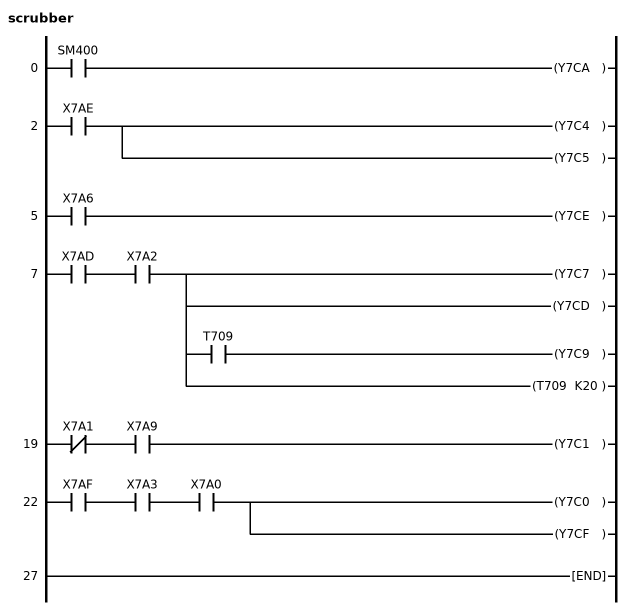
[picture p192: ladder of scrubber, rungs at steps 0 to 27]
0     LD      SM400
      OUT     Y7CA
2     LD      X7AE
      OUT     Y7C4
      OUT     Y7C5
5     LD      X7A6
      OUT     Y7CE
7     LD      X7AD
      AND     X7A2
      OUT     Y7C7
      OUT     Y7CD
      MPS
      AND     T709
      OUT     Y7C9
      MPP
      OUT     T709 K20
19    LDI     X7A1
      AND     X7A9
      OUT     Y7C1
22    LD      X7AF
      AND     X7A3
      AND     X7A0
      OUT     Y7C0
      OUT     Y7CF
27    END
END_PROGRAM

PROGRAM send_to_c
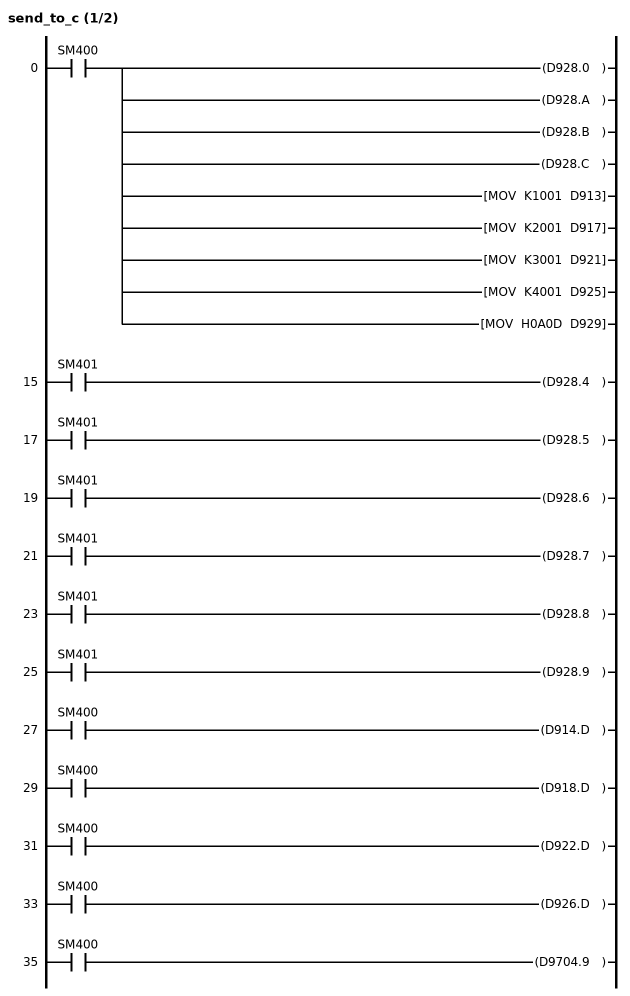
0     LD      SM400
      OUT     D928.0
      OUT     D928.A
      OUT     D928.B
      OUT     D928.C
      MOV     K1001 D913
      MOV     K2001 D917
      MOV     K3001 D921
      MOV     K4001 D925
      MOV     H0A0D D929
15    LD      SM401
      OUT     D928.4
17    LD      SM401
      OUT     D928.5
19    LD      SM401
      OUT     D928.6
21    LD      SM401
      OUT     D928.7
23    LD      SM401
      OUT     D928.8
25    LD      SM401
      OUT     D928.9
27    LD      SM400
      OUT     D914.D
29    LD      SM400
      OUT     D918.D
31    LD      SM400
      OUT     D922.D
33    LD      SM400
      OUT     D926.D
35    LD      SM400
      OUT     D9704.9
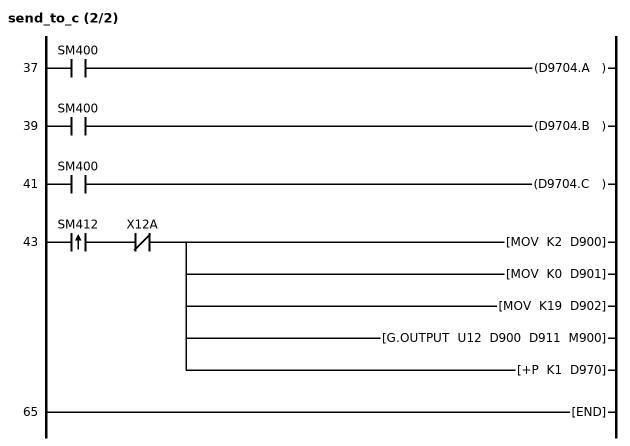
37    LD      SM400
      OUT     D9704.A
39    LD      SM400
      OUT     D9704.B
41    LD      SM400
      OUT     D9704.C
43    LDP     SM412
      ANI     X12A
      MOV     K2 D900
      MOV     K0 D901
      MOV     K19 D902
      G.OUTPUT U12 D900 D911 M900
      +P      K1 D970
65    END
END_PROGRAM

PROGRAM shower
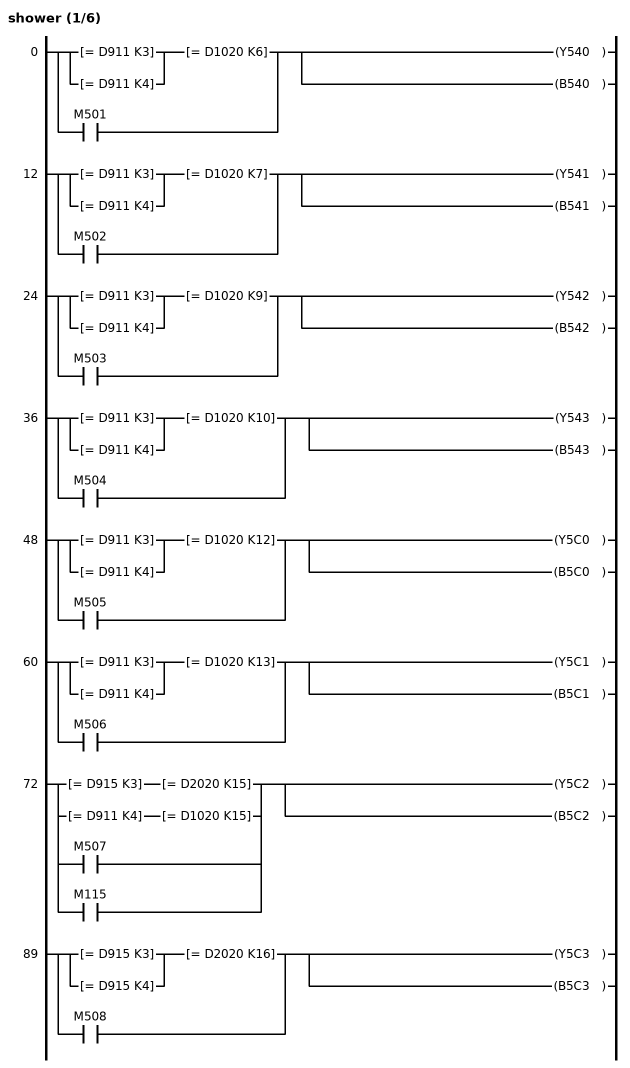
0     LD=     D911 K3
      OR=     D911 K4
      AND=    D1020 K6
      OR      M501
      OUT     Y540
      OUT     B540
12    LD=     D911 K3
      OR=     D911 K4
      AND=    D1020 K7
      OR      M502
      OUT     Y541
      OUT     B541
24    LD=     D911 K3
      OR=     D911 K4
      AND=    D1020 K9
      OR      M503
      OUT     Y542
      OUT     B542
36    LD=     D911 K3
      OR=     D911 K4
      AND=    D1020 K10
      OR      M504
      OUT     Y543
      OUT     B543
48    LD=     D911 K3
      OR=     D911 K4
      AND=    D1020 K12
      OR      M505
      OUT     Y5C0
      OUT     B5C0
60    LD=     D911 K3
      OR=     D911 K4
      AND=    D1020 K13
      OR      M506
      OUT     Y5C1
      OUT     B5C1
72    LD=     D915 K3
      AND=    D2020 K15
      LD=     D911 K4
      AND=    D1020 K15
      ORB
      OR      M507
      OR      M115
      OUT     Y5C2
      OUT     B5C2
89    LD=     D915 K3
      OR=     D915 K4
      AND=    D2020 K16
      OR      M508
      OUT     Y5C3
      OUT     B5C3
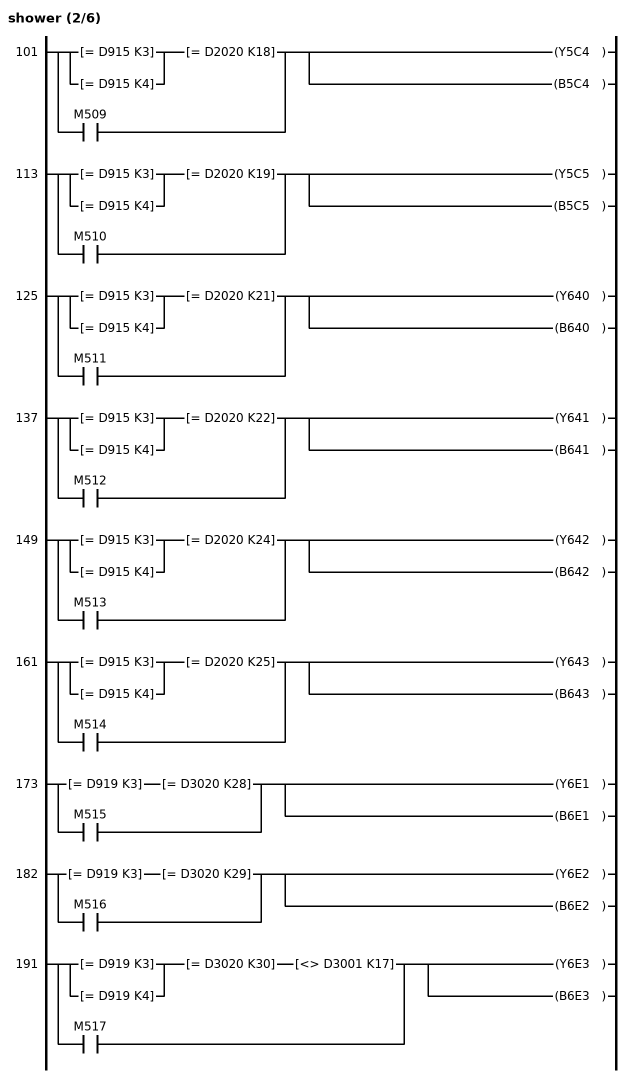
101   LD=     D915 K3
      OR=     D915 K4
      AND=    D2020 K18
      OR      M509
      OUT     Y5C4
      OUT     B5C4
113   LD=     D915 K3
      OR=     D915 K4
      AND=    D2020 K19
      OR      M510
      OUT     Y5C5
      OUT     B5C5
125   LD=     D915 K3
      OR=     D915 K4
      AND=    D2020 K21
      OR      M511
      OUT     Y640
      OUT     B640
137   LD=     D915 K3
      OR=     D915 K4
      AND=    D2020 K22
      OR      M512
      OUT     Y641
      OUT     B641
149   LD=     D915 K3
      OR=     D915 K4
      AND=    D2020 K24
      OR      M513
      OUT     Y642
      OUT     B642
161   LD=     D915 K3
      OR=     D915 K4
      AND=    D2020 K25
      OR      M514
      OUT     Y643
      OUT     B643
173   LD=     D919 K3
      AND=    D3020 K28
      OR      M515
      OUT     Y6E1
      OUT     B6E1
182   LD=     D919 K3
      AND=    D3020 K29
      OR      M516
      OUT     Y6E2
      OUT     B6E2
191   LD=     D919 K3
      OR=     D919 K4
      AND=    D3020 K30
      AND<>   D3001 K17
      OR      M517
      OUT     Y6E3
      OUT     B6E3
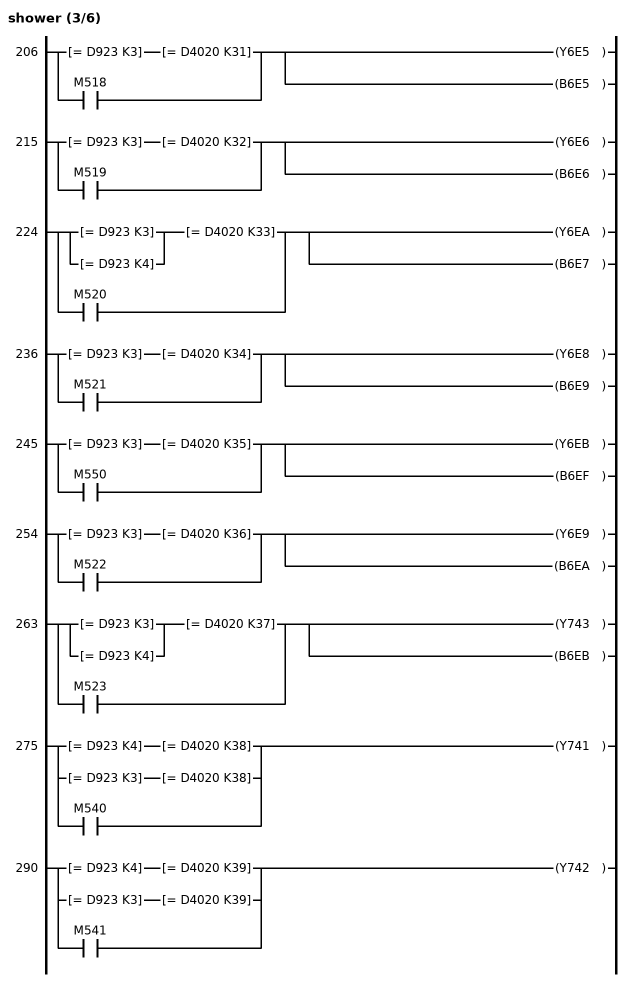
206   LD=     D923 K3
      AND=    D4020 K31
      OR      M518
      OUT     Y6E5
      OUT     B6E5
215   LD=     D923 K3
      AND=    D4020 K32
      OR      M519
      OUT     Y6E6
      OUT     B6E6
224   LD=     D923 K3
      OR=     D923 K4
      AND=    D4020 K33
      OR      M520
      OUT     Y6EA
      OUT     B6E7
236   LD=     D923 K3
      AND=    D4020 K34
      OR      M521
      OUT     Y6E8
      OUT     B6E9
245   LD=     D923 K3
      AND=    D4020 K35
      OR      M550
      OUT     Y6EB
      OUT     B6EF
254   LD=     D923 K3
      AND=    D4020 K36
      OR      M522
      OUT     Y6E9
      OUT     B6EA
263   LD=     D923 K3
      OR=     D923 K4
      AND=    D4020 K37
      OR      M523
      OUT     Y743
      OUT     B6EB
275   LD=     D923 K4
      AND=    D4020 K38
      LD=     D923 K3
      AND=    D4020 K38
      ORB
      OR      M540
      OUT     Y741
290   LD=     D923 K4
      AND=    D4020 K39
      LD=     D923 K3
      AND=    D4020 K39
      ORB
      OR      M541
      OUT     Y742
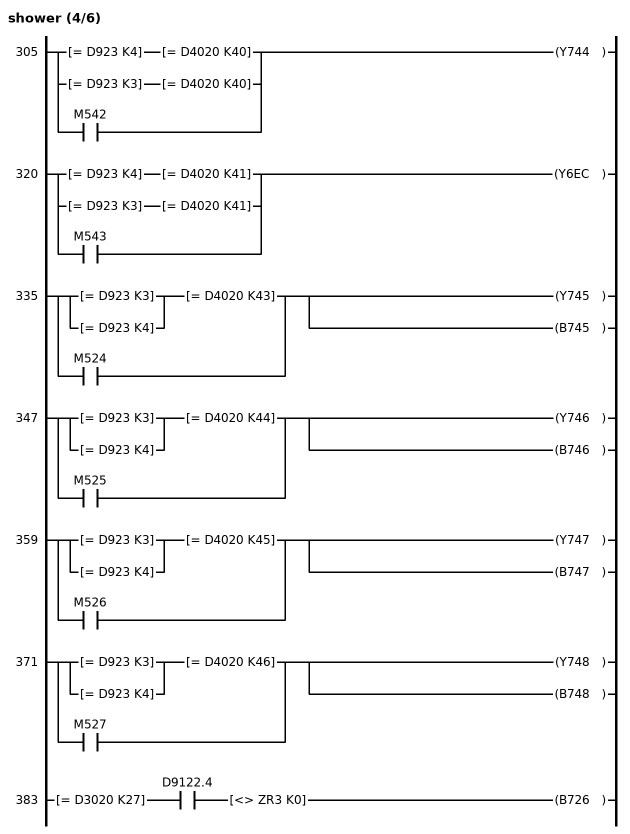
305   LD=     D923 K4
      AND=    D4020 K40
      LD=     D923 K3
      AND=    D4020 K40
      ORB
      OR      M542
      OUT     Y744
320   LD=     D923 K4
      AND=    D4020 K41
      LD=     D923 K3
      AND=    D4020 K41
      ORB
      OR      M543
      OUT     Y6EC
335   LD=     D923 K3
      OR=     D923 K4
      AND=    D4020 K43
      OR      M524
      OUT     Y745
      OUT     B745
347   LD=     D923 K3
      OR=     D923 K4
      AND=    D4020 K44
      OR      M525
      OUT     Y746
      OUT     B746
359   LD=     D923 K3
      OR=     D923 K4
      AND=    D4020 K45
      OR      M526
      OUT     Y747
      OUT     B747
371   LD=     D923 K3
      OR=     D923 K4
      AND=    D4020 K46
      OR      M527
      OUT     Y748
      OUT     B748
383   LD=     D3020 K27
      AND     D9122.4
      AND<>   ZR3 K0
      OUT     B726
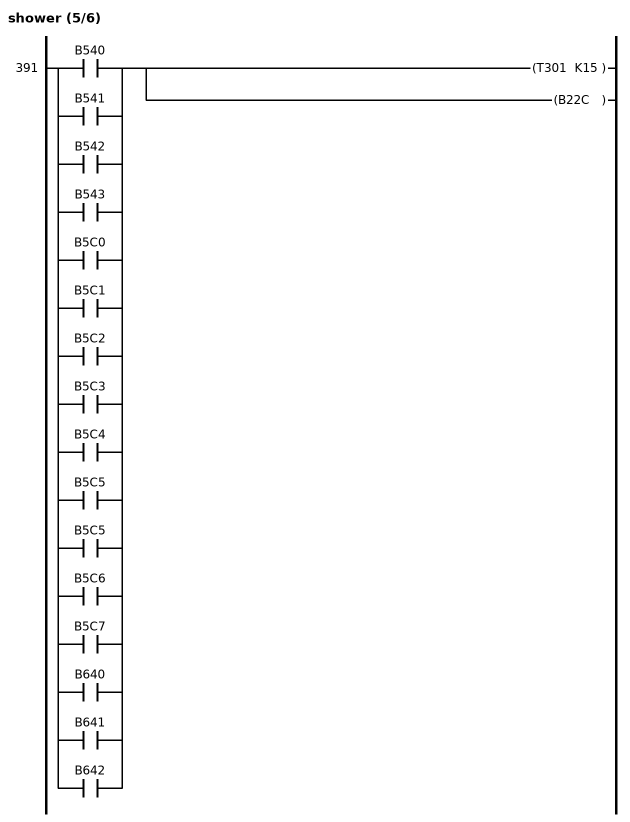
391   LD      B540
      OR      B541
      OR      B542
      OR      B543
      OR      B5C0
      OR      B5C1
      OR      B5C2
      OR      B5C3
      OR      B5C4
      OR      B5C5
      OR      B5C5
      OR      B5C6
      OR      B5C7
      OR      B640
      OR      B641
      OR      B642
      OUT     T301 K15
      OUT     B22C
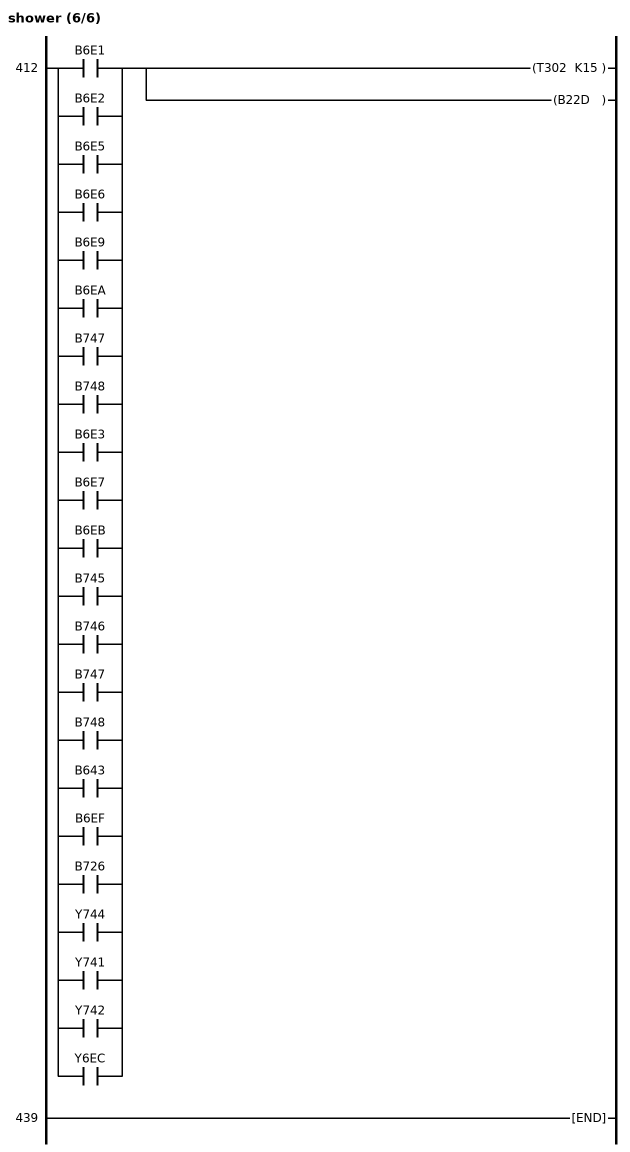
412   LD      B6E1
      OR      B6E2
      OR      B6E5
      OR      B6E6
      OR      B6E9
      OR      B6EA
      OR      B747
      OR      B748
      OR      B6E3
      OR      B6E7
      OR      B6EB
      OR      B745
      OR      B746
      OR      B747
      OR      B748
      OR      B643
      OR      B6EF
      OR      B726
      OR      Y744
      OR      Y741
      OR      Y742
      OR      Y6EC
      OUT     T302 K15
      OUT     B22D
439   END
END_PROGRAM

PROGRAM Start_cycle
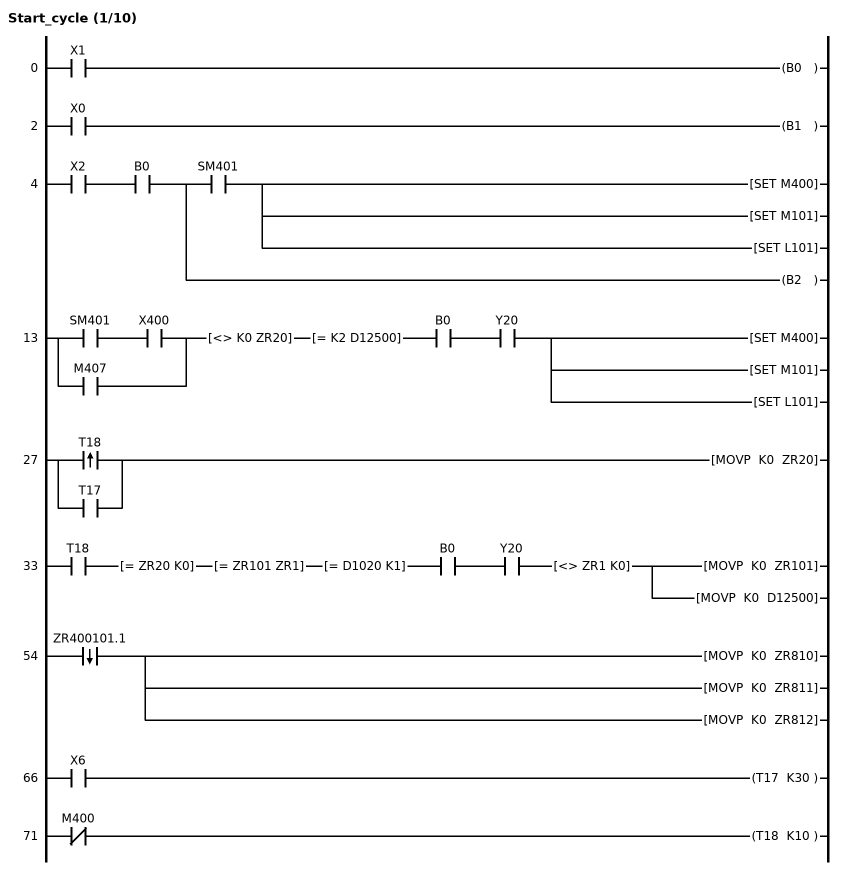
0     LD      X1
      OUT     B0
2     LD      X0
      OUT     B1
4     LD      X2
      AND     B0
      MPS
      AND     SM401
      SET     M400
      SET     M101
      SET     L101
      MPP
      OUT     B2
13    LD      SM401
      AND     X400
      OR      M407
      AND<>   K0 ZR20
      AND=    K2 D12500
      AND     B0
      AND     Y20
      SET     M400
      SET     M101
      SET     L101
27    LDP     T18
      OR      T17
      MOVP    K0 ZR20
33    LD      T18
      AND=    ZR20 K0
      AND=    ZR101 ZR1
      AND=    D1020 K1
      AND     B0
      AND     Y20
      AND<>   ZR1 K0
      MOVP    K0 ZR101
      MOVP    K0 D12500
54    LDF     ZR400101.1
      MOVP    K0 ZR810
      MOVP    K0 ZR811
      MOVP    K0 ZR812
66    LD      X6
      OUT     T17 K30
71    LDI     M400
      OUT     T18 K10
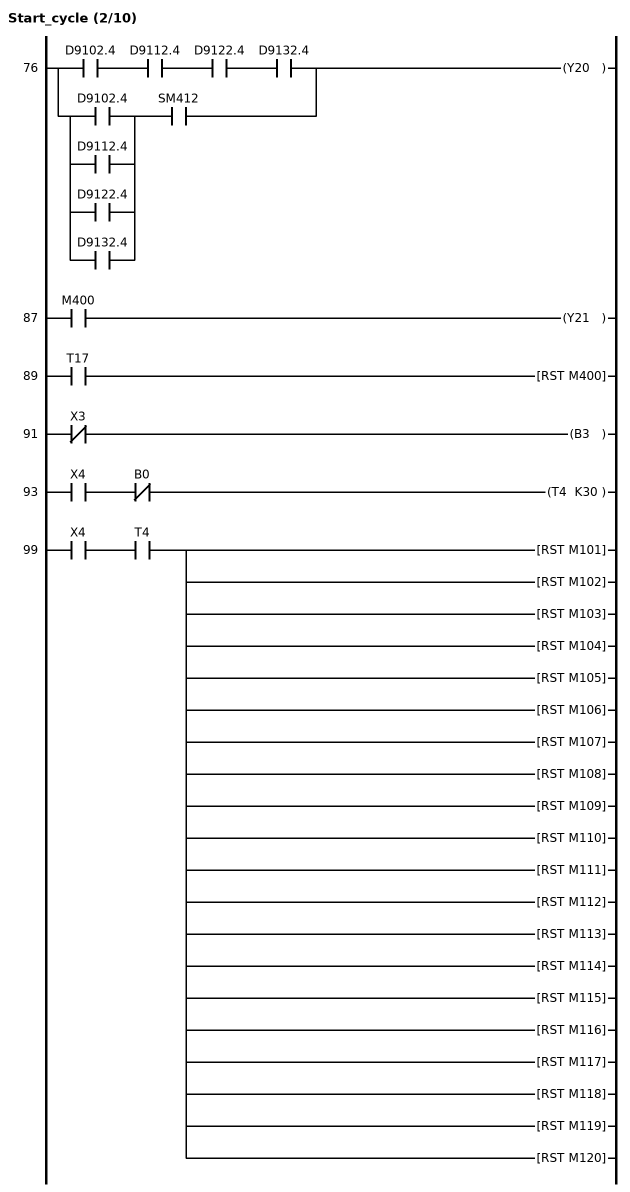
76    LD      D9102.4
      AND     D9112.4
      AND     D9122.4
      AND     D9132.4
      LD      D9102.4
      OR      D9112.4
      OR      D9122.4
      OR      D9132.4
      AND     SM412
      ORB
      OUT     Y20
87    LD      M400
      OUT     Y21
89    LD      T17
      RST     M400
91    LDI     X3
      OUT     B3
93    LD      X4
      ANI     B0
      OUT     T4 K30
99    LD      X4
      AND     T4
      RST     M101
      RST     M102
      RST     M103
      RST     M104
      RST     M105
      RST     M106
      RST     M107
      RST     M108
      RST     M109
      RST     M110
      RST     M111
      RST     M112
      RST     M113
      RST     M114
      RST     M115
      RST     M116
      RST     M117
      RST     M118
      RST     M119
      RST     M120
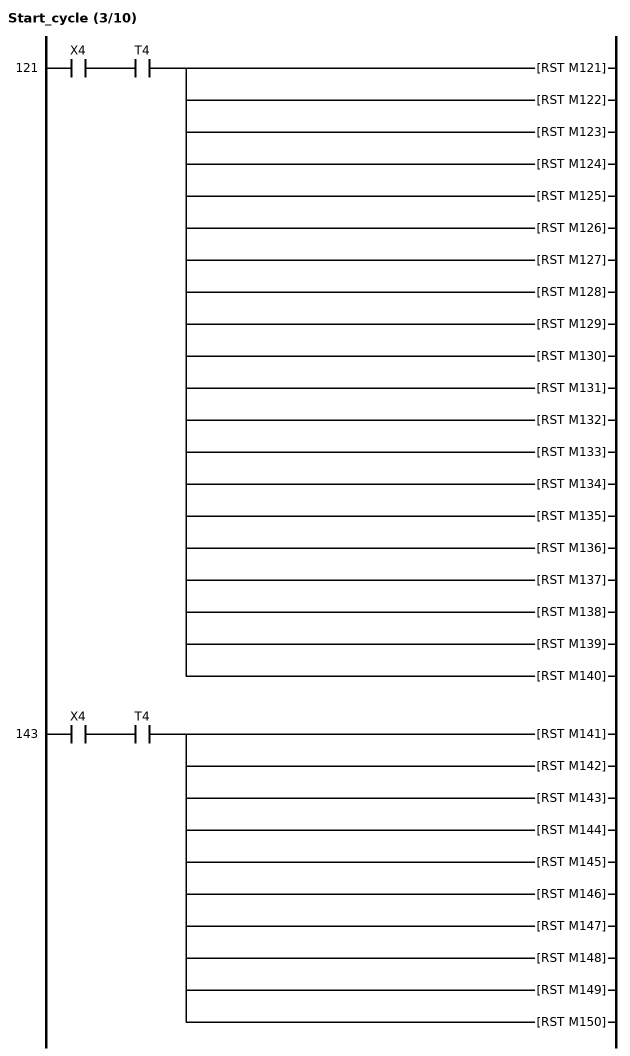
121   LD      X4
      AND     T4
      RST     M121
      RST     M122
      RST     M123
      RST     M124
      RST     M125
      RST     M126
      RST     M127
      RST     M128
      RST     M129
      RST     M130
      RST     M131
      RST     M132
      RST     M133
      RST     M134
      RST     M135
      RST     M136
      RST     M137
      RST     M138
      RST     M139
      RST     M140
143   LD      X4
      AND     T4
      RST     M141
      RST     M142
      RST     M143
      RST     M144
      RST     M145
      RST     M146
      RST     M147
      RST     M148
      RST     M149
      RST     M150
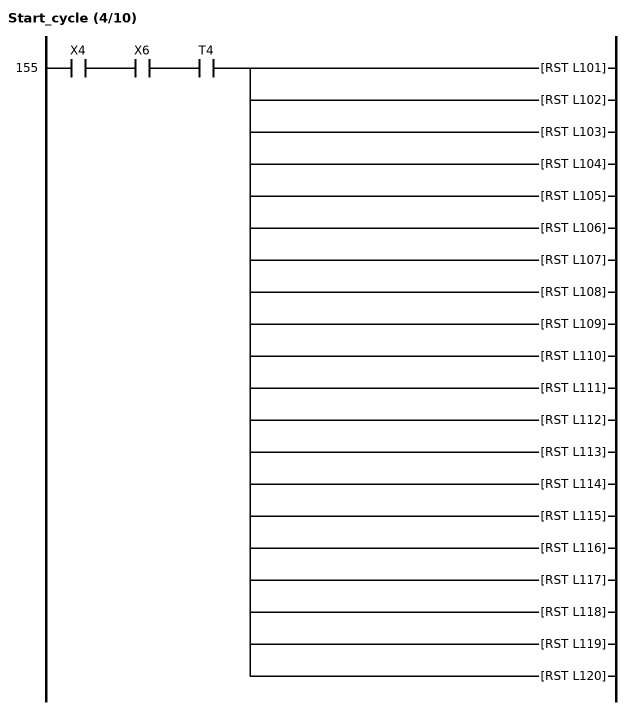
155   LD      X4
      AND     X6
      AND     T4
      RST     L101
      RST     L102
      RST     L103
      RST     L104
      RST     L105
      RST     L106
      RST     L107
      RST     L108
      RST     L109
      RST     L110
      RST     L111
      RST     L112
      RST     L113
      RST     L114
      RST     L115
      RST     L116
      RST     L117
      RST     L118
      RST     L119
      RST     L120
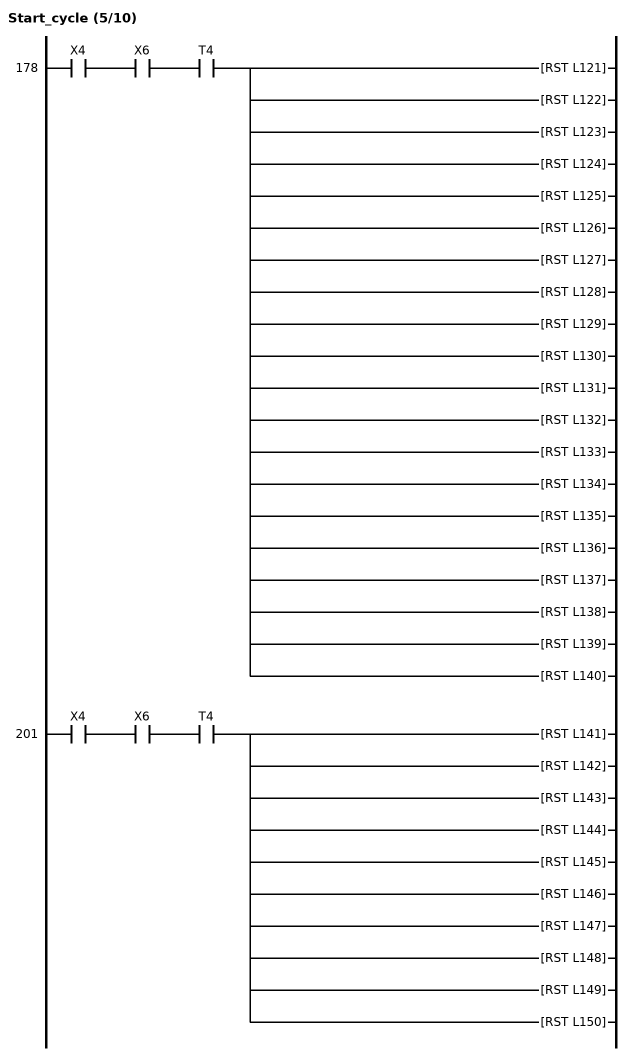
178   LD      X4
      AND     X6
      AND     T4
      RST     L121
      RST     L122
      RST     L123
      RST     L124
      RST     L125
      RST     L126
      RST     L127
      RST     L128
      RST     L129
      RST     L130
      RST     L131
      RST     L132
      RST     L133
      RST     L134
      RST     L135
      RST     L136
      RST     L137
      RST     L138
      RST     L139
      RST     L140
201   LD      X4
      AND     X6
      AND     T4
      RST     L141
      RST     L142
      RST     L143
      RST     L144
      RST     L145
      RST     L146
      RST     L147
      RST     L148
      RST     L149
      RST     L150
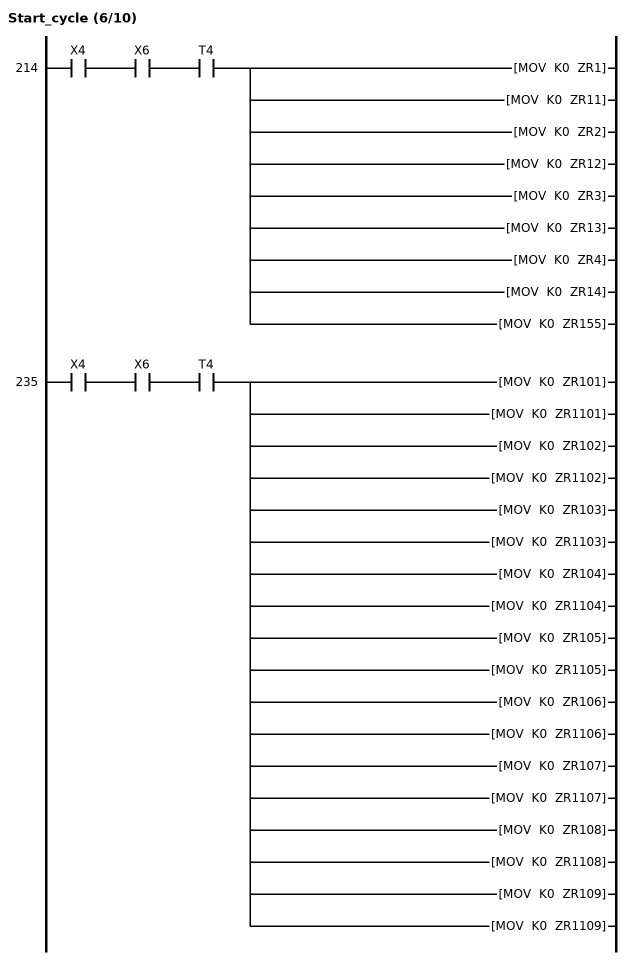
214   LD      X4
      AND     X6
      AND     T4
      MOV     K0 ZR1
      MOV     K0 ZR11
      MOV     K0 ZR2
      MOV     K0 ZR12
      MOV     K0 ZR3
      MOV     K0 ZR13
      MOV     K0 ZR4
      MOV     K0 ZR14
      MOV     K0 ZR155
235   LD      X4
      AND     X6
      AND     T4
      MOV     K0 ZR101
      MOV     K0 ZR1101
      MOV     K0 ZR102
      MOV     K0 ZR1102
      MOV     K0 ZR103
      MOV     K0 ZR1103
      MOV     K0 ZR104
      MOV     K0 ZR1104
      MOV     K0 ZR105
      MOV     K0 ZR1105
      MOV     K0 ZR106
      MOV     K0 ZR1106
      MOV     K0 ZR107
      MOV     K0 ZR1107
      MOV     K0 ZR108
      MOV     K0 ZR1108
      MOV     K0 ZR109
      MOV     K0 ZR1109
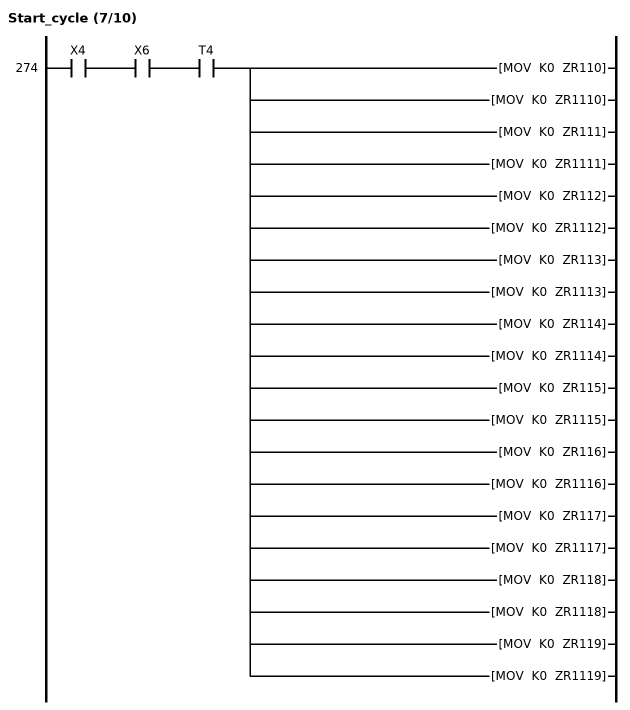
274   LD      X4
      AND     X6
      AND     T4
      MOV     K0 ZR110
      MOV     K0 ZR1110
      MOV     K0 ZR111
      MOV     K0 ZR1111
      MOV     K0 ZR112
      MOV     K0 ZR1112
      MOV     K0 ZR113
      MOV     K0 ZR1113
      MOV     K0 ZR114
      MOV     K0 ZR1114
      MOV     K0 ZR115
      MOV     K0 ZR1115
      MOV     K0 ZR116
      MOV     K0 ZR1116
      MOV     K0 ZR117
      MOV     K0 ZR1117
      MOV     K0 ZR118
      MOV     K0 ZR1118
      MOV     K0 ZR119
      MOV     K0 ZR1119
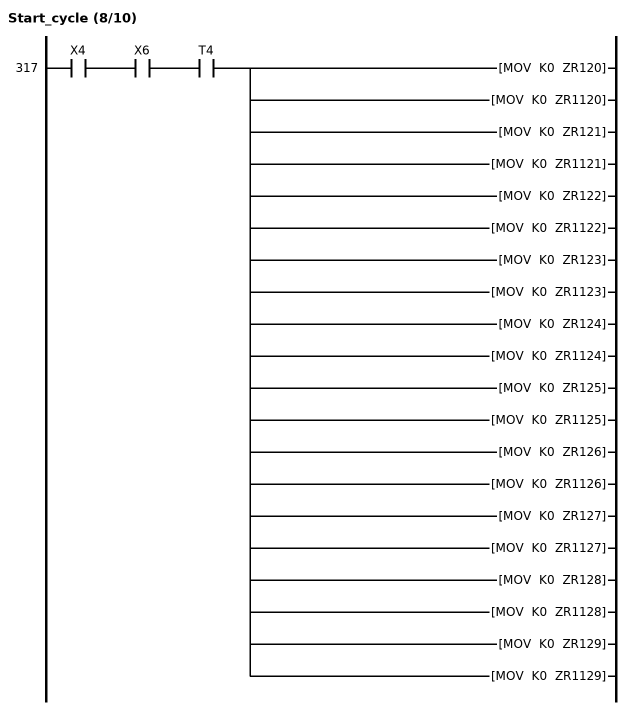
317   LD      X4
      AND     X6
      AND     T4
      MOV     K0 ZR120
      MOV     K0 ZR1120
      MOV     K0 ZR121
      MOV     K0 ZR1121
      MOV     K0 ZR122
      MOV     K0 ZR1122
      MOV     K0 ZR123
      MOV     K0 ZR1123
      MOV     K0 ZR124
      MOV     K0 ZR1124
      MOV     K0 ZR125
      MOV     K0 ZR1125
      MOV     K0 ZR126
      MOV     K0 ZR1126
      MOV     K0 ZR127
      MOV     K0 ZR1127
      MOV     K0 ZR128
      MOV     K0 ZR1128
      MOV     K0 ZR129
      MOV     K0 ZR1129
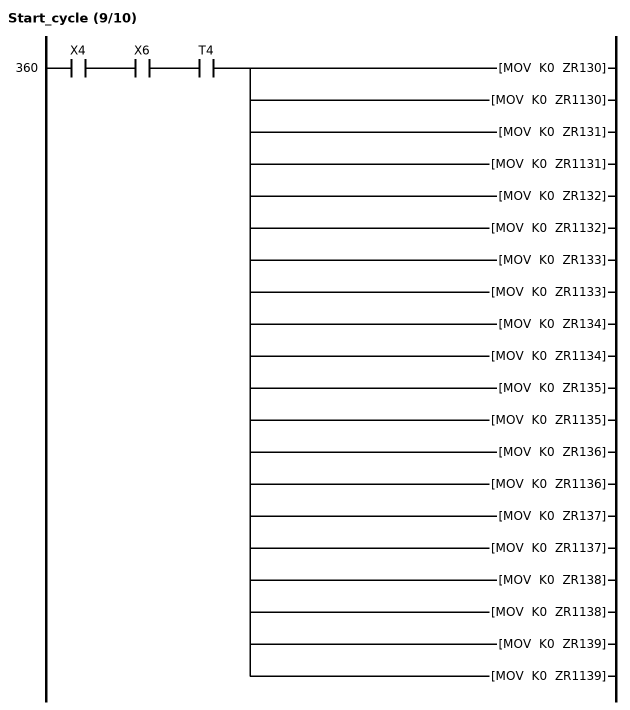
360   LD      X4
      AND     X6
      AND     T4
      MOV     K0 ZR130
      MOV     K0 ZR1130
      MOV     K0 ZR131
      MOV     K0 ZR1131
      MOV     K0 ZR132
      MOV     K0 ZR1132
      MOV     K0 ZR133
      MOV     K0 ZR1133
      MOV     K0 ZR134
      MOV     K0 ZR1134
      MOV     K0 ZR135
      MOV     K0 ZR1135
      MOV     K0 ZR136
      MOV     K0 ZR1136
      MOV     K0 ZR137
      MOV     K0 ZR1137
      MOV     K0 ZR138
      MOV     K0 ZR1138
      MOV     K0 ZR139
      MOV     K0 ZR1139
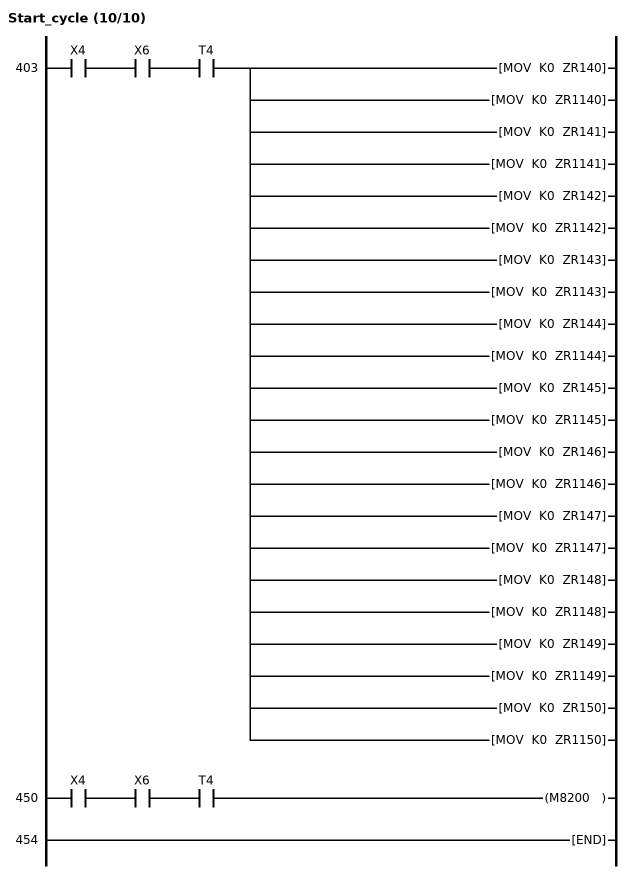
403   LD      X4
      AND     X6
      AND     T4
      MOV     K0 ZR140
      MOV     K0 ZR1140
      MOV     K0 ZR141
      MOV     K0 ZR1141
      MOV     K0 ZR142
      MOV     K0 ZR1142
      MOV     K0 ZR143
      MOV     K0 ZR1143
      MOV     K0 ZR144
      MOV     K0 ZR1144
      MOV     K0 ZR145
      MOV     K0 ZR1145
      MOV     K0 ZR146
      MOV     K0 ZR1146
      MOV     K0 ZR147
      MOV     K0 ZR1147
      MOV     K0 ZR148
      MOV     K0 ZR1148
      MOV     K0 ZR149
      MOV     K0 ZR1149
      MOV     K0 ZR150
      MOV     K0 ZR1150
450   LD      X4
      AND     X6
      AND     T4
      OUT     M8200
454   END
END_PROGRAM

PROGRAM start_WR
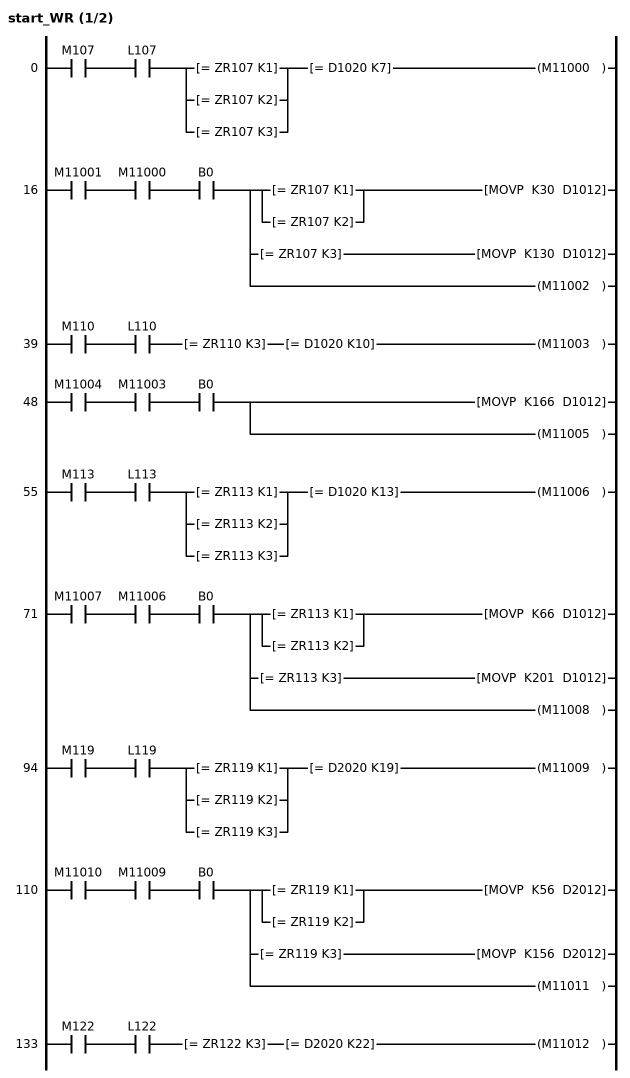
0     LD      M107
      AND     L107
      LD=     ZR107 K1
      OR=     ZR107 K2
      OR=     ZR107 K3
      ANB
      AND=    D1020 K7
      OUT     M11000
16    LD      M11001
      AND     M11000
      AND     B0
      MPS
      LD=     ZR107 K1
      OR=     ZR107 K2
      ANB
      MOVP    K30 D1012
      MRD
      AND=    ZR107 K3
      MOVP    K130 D1012
      MPP
      OUT     M11002
39    LD      M110
      AND     L110
      AND=    ZR110 K3
      AND=    D1020 K10
      OUT     M11003
48    LD      M11004
      AND     M11003
      AND     B0
      MOVP    K166 D1012
      OUT     M11005
55    LD      M113
      AND     L113
      LD=     ZR113 K1
      OR=     ZR113 K2
      OR=     ZR113 K3
      ANB
      AND=    D1020 K13
      OUT     M11006
71    LD      M11007
      AND     M11006
      AND     B0
      MPS
      LD=     ZR113 K1
      OR=     ZR113 K2
      ANB
      MOVP    K66 D1012
      MRD
      AND=    ZR113 K3
      MOVP    K201 D1012
      MPP
      OUT     M11008
94    LD      M119
      AND     L119
      LD=     ZR119 K1
      OR=     ZR119 K2
      OR=     ZR119 K3
      ANB
      AND=    D2020 K19
      OUT     M11009
110   LD      M11010
      AND     M11009
      AND     B0
      MPS
      LD=     ZR119 K1
      OR=     ZR119 K2
      ANB
      MOVP    K56 D2012
      MRD
      AND=    ZR119 K3
      MOVP    K156 D2012
      MPP
      OUT     M11011
133   LD      M122
      AND     L122
      AND=    ZR122 K3
      AND=    D2020 K22
      OUT     M11012
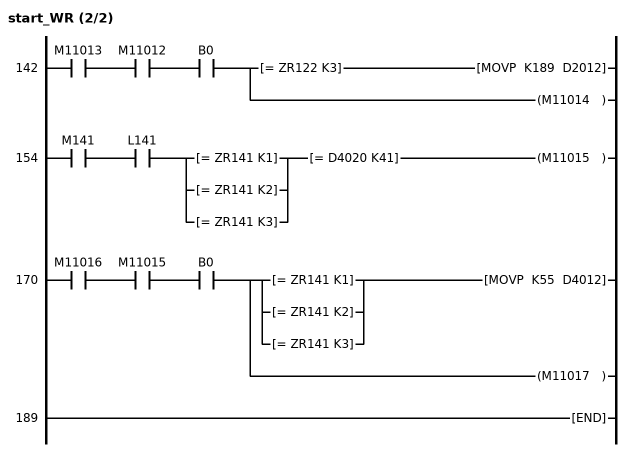
142   LD      M11013
      AND     M11012
      AND     B0
      MPS
      AND=    ZR122 K3
      MOVP    K189 D2012
      MPP
      OUT     M11014
154   LD      M141
      AND     L141
      LD=     ZR141 K1
      OR=     ZR141 K2
      OR=     ZR141 K3
      ANB
      AND=    D4020 K41
      OUT     M11015
170   LD      M11016
      AND     M11015
      AND     B0
      MPS
      LD=     ZR141 K1
      OR=     ZR141 K2
      OR=     ZR141 K3
      ANB
      MOVP    K55 D4012
      MPP
      OUT     M11017
189   END
END_PROGRAM

FUNCTION_BLOCK tank_PV
VAR_INPUT
  ON_BY_ORDER : BOOL;
  Stay_ON : BOOL;
  Reset_0 : BOOL;
END_VAR
VAR_OUTPUT
  PV : INT;
END_VAR
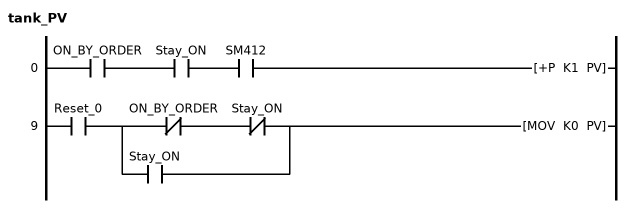
0     LD      ON_BY_ORDER
      AND     Stay_ON
      AND     SM412
      +P      K1 PV
9     LD      Reset_0
      LDI     ON_BY_ORDER
      ANI     Stay_ON
      OR      Stay_ON
      ANB
      MOV     K0 PV
END_FUNCTION_BLOCK

PROGRAM tank_time_A
VAR
  tank_PV_2 : tank_PV;
  tank_PV_3 : tank_PV;
  tank_PV_4 : tank_PV;
  tank_PV_5 : tank_PV;
  tank_PV_6 : tank_PV;
  tank_PV_7 : tank_PV;
  tank_PV_8 : tank_PV;
  tank_PV_9 : tank_PV;
  tank_PV_10 : tank_PV;
  tank_PV_11 : tank_PV;
  tank_PV_12 : tank_PV;
  tank_PV_13 : tank_PV;
  tank_PV_14 : tank_PV;
  tank_PV_15 : tank_PV;
  tank_PV_16 : tank_PV;
  tank_PV_17 : tank_PV;
  tank_PV_18 : tank_PV;
  tank_PV_19 : tank_PV;
  tank_PV_21 : tank_PV;
  tank_PV_22 : tank_PV;
  tank_PV_20 : tank_PV;
  tank_PV_23 : tank_PV;
  tank_PV_24 : tank_PV;
  tank_PV_25 : tank_PV;
  tank_PV_26 : tank_PV;
  tank_PV_27 : tank_PV;
  tank_PV_28 : tank_PV;
  tank_PV_29 : tank_PV;
  tank_PV_30 : tank_PV;
  tank_PV_31 : tank_PV;
  tank_PV_32 : tank_PV;
  tank_PV_33 : tank_PV;
  tank_PV_34 : tank_PV;
  tank_PV_35 : tank_PV;
  tank_PV_36 : tank_PV;
  tank_PV_37 : tank_PV;
  tank_PV_38 : tank_PV;
  tank_PV_39 : tank_PV;
  tank_PV_40 : tank_PV;
  tank_PV_41 : tank_PV;
  tank_PV_42 : tank_PV;
  tank_PV_43 : tank_PV;
  tank_PV_44 : tank_PV;
  tank_PV_45 : tank_PV;
  tank_PV_46 : tank_PV;
  tank_PV_47 : tank_PV;
  tank_PV_48 : tank_PV;
  tank_PV_49 : tank_PV;
  tank_PV_50 : tank_PV;
END_VAR
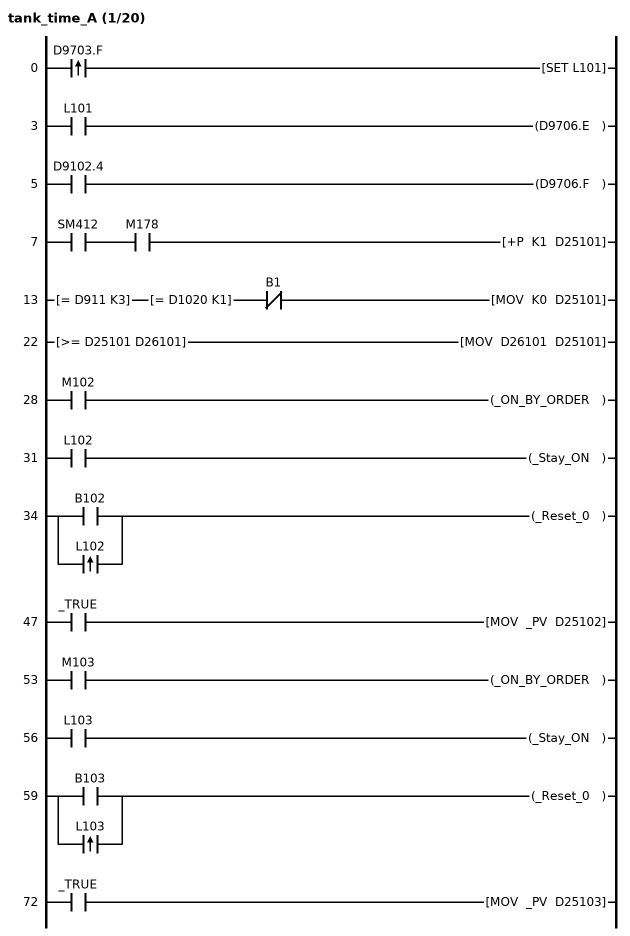
0     LDP     D9703.F
      SET     L101
3     LD      L101
      OUT     D9706.E
5     LD      D9102.4
      OUT     D9706.F
7     LD      SM412
      AND     M178
      +P      K1 D25101
13    LD=     D911 K3
      AND=    D1020 K1
      ANI     B1
      MOV     K0 D25101
22    LD>=    D25101 D26101
      MOV     D26101 D25101
; FB BLK START tank_PV(tank_PV_2)
28    LD      M102
      OUT     _ON_BY_ORDER
31    LD      L102
      OUT     _Stay_ON
34    LD      B102
      ORP     L102
      OUT     _Reset_0
; FB START
; FB_NAME tank_PV
; INSTANCE_NAME tank_PV_2
; FB IN_B:ON_BY_ORDER
; FB OUT_PV:W
; FB IN_B:Stay_ON
; FB IN_B:Reset_0
; FB END
47    LD      _TRUE
      MOV     _PV D25102
; FB BLK END
; FB BLK START tank_PV(tank_PV_3)
53    LD      M103
      OUT     _ON_BY_ORDER
56    LD      L103
      OUT     _Stay_ON
59    LD      B103
      ORP     L103
      OUT     _Reset_0
; FB START
; FB_NAME tank_PV
; INSTANCE_NAME tank_PV_3
; FB IN_B:ON_BY_ORDER
; FB OUT_PV:W
; FB IN_B:Stay_ON
; FB IN_B:Reset_0
; FB END
72    LD      _TRUE
      MOV     _PV D25103
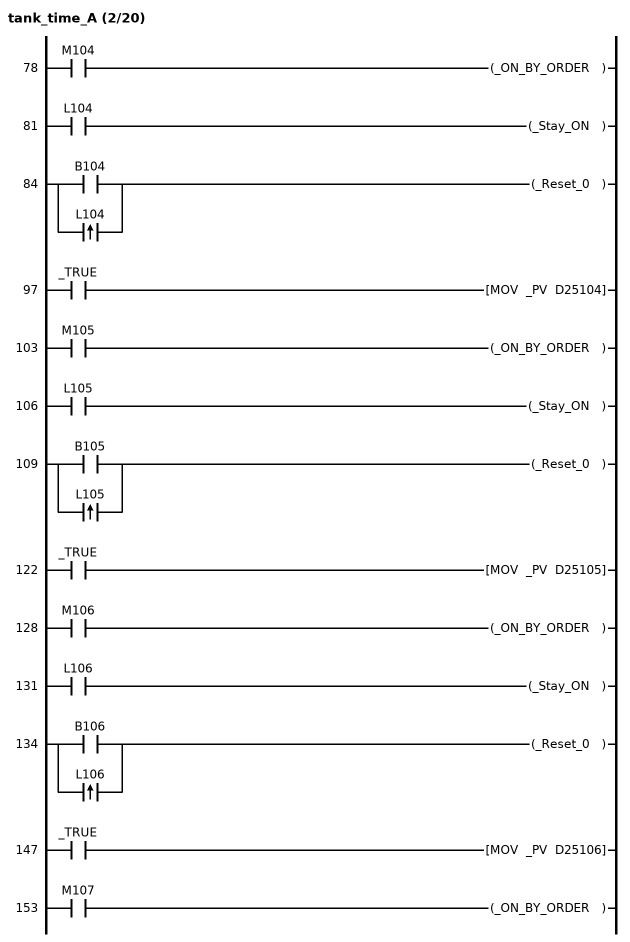
; FB BLK END
; FB BLK START tank_PV(tank_PV_4)
78    LD      M104
      OUT     _ON_BY_ORDER
81    LD      L104
      OUT     _Stay_ON
84    LD      B104
      ORP     L104
      OUT     _Reset_0
; FB START
; FB_NAME tank_PV
; INSTANCE_NAME tank_PV_4
; FB IN_B:ON_BY_ORDER
; FB OUT_PV:W
; FB IN_B:Stay_ON
; FB IN_B:Reset_0
; FB END
97    LD      _TRUE
      MOV     _PV D25104
; FB BLK END
; FB BLK START tank_PV(tank_PV_5)
103   LD      M105
      OUT     _ON_BY_ORDER
106   LD      L105
      OUT     _Stay_ON
109   LD      B105
      ORP     L105
      OUT     _Reset_0
; FB START
; FB_NAME tank_PV
; INSTANCE_NAME tank_PV_5
; FB IN_B:ON_BY_ORDER
; FB OUT_PV:W
; FB IN_B:Stay_ON
; FB IN_B:Reset_0
; FB END
122   LD      _TRUE
      MOV     _PV D25105
; FB BLK END
; FB BLK START tank_PV(tank_PV_6)
128   LD      M106
      OUT     _ON_BY_ORDER
131   LD      L106
      OUT     _Stay_ON
134   LD      B106
      ORP     L106
      OUT     _Reset_0
; FB START
; FB_NAME tank_PV
; INSTANCE_NAME tank_PV_6
; FB IN_B:ON_BY_ORDER
; FB OUT_PV:W
; FB IN_B:Stay_ON
; FB IN_B:Reset_0
; FB END
147   LD      _TRUE
      MOV     _PV D25106
; FB BLK END
; FB BLK START tank_PV(tank_PV_7)
153   LD      M107
      OUT     _ON_BY_ORDER
